{attribute 'linkalways'} 
{attribute 'no_explicit_call' := 'This FB is a CLASS and must be accessed using methods or properties'}
{attribute 'enable_dynamic_creation'}
FUNCTION_BLOCK GetBlueprintsRpcHandler IMPLEMENTS I_RpcHandler
VAR
	nodePrototypes : I_NodePrototypes;
END_VAR

METHOD FB_init : BOOL
VAR_INPUT
	bInitRetains : BOOL; // if TRUE, the retain variables are initialized (warm start / cold start)
	bInCopyCode : BOOL;  // if TRUE, the instance afterwards gets moved into the copy code (online change)
	NodePrototypes : I_NodePrototypes;
END_VAR
this^.nodePrototypes := NodePrototypes;
END_METHOD

METHOD Handle
VAR_INPUT
	Parameters : I_Deserializer;
	Response : I_SynchronousRpcResponse;
END_VAR
IF nodePrototypes = 0 THEN
	Response.RejectWithMessage('GetBlueprintsRpcHandler has not been initialized with a valid nodePrototypes object');
	RETURN;
END_IF

Response.CompleteWithObject(nodePrototypes);
END_METHOD

METHOD PUBLIC Initialize
VAR_INPUT
	NodePrototypes : I_NodePrototypes;
END_VAR
this^.nodePrototypes := NodePrototypes;
END_METHOD

END_FUNCTION_BLOCK

(* stored: Version 1.1.0.1, ProductVersion 3.1.4024.12
   POU GetBlueprintsRpcHandler: Id {5f1261a8-a78b-47cb-8ce3-4f6764554f1c}, SpecialFunc None
   Folder Constructor: Id {4153f967-c5de-4128-a5d1-9198f1228c47}
   Method FB_init: Id {ceef250b-d580-479c-a4e6-db612b691818}
   Method Handle: Id {27315dcd-2d70-4147-9721-52dd88a1612b}
   Method Initialize: Id {9ad671d0-ce42-4ff2-977f-33468cbea023} *)
